// Block: AccRollConveyor_PERS

DATA_BLOCK AccRollConveyor_PERS
VERSION : 0.1
   NON_RETAIN
   VAR
      PersistentValues : udt_AccRollConveyor_Pers;
   END_VAR

BEGIN
   // No initialization required
END_DATA_BLOCK
